FUNCTION_BLOCK FB_CalculateDiamondThickness
VAR
END_VAR


METHOD PUBLIC Calculate
VAR_INPUT
    fDesiredTransmission : LREAL; // [1]
    fPhotonEnergy : LREAL; // [eV]
END_VAR
VAR_OUTPUT
    fThickness : LREAL; // [mm]
END_VAR
END_METHOD

END_FUNCTION_BLOCK

(* stored: Version 1.1.0.1
   POU FB_CalculateDiamondThickness: Id {bc9bfacc-7d3a-4611-b219-338ca75019df}, SpecialFunc None
   Method Calculate: Id {bf69efd6-1e63-4e72-bb10-5ffc888b9575} *)
